SYSTEM temexdmod2
  (* Version 1.0, Author, 4DIAC-Consortium *)
  APPLICATION plantwide
  END_APPLICATION
  APPLICATION App1_ProdQualityandConstraints
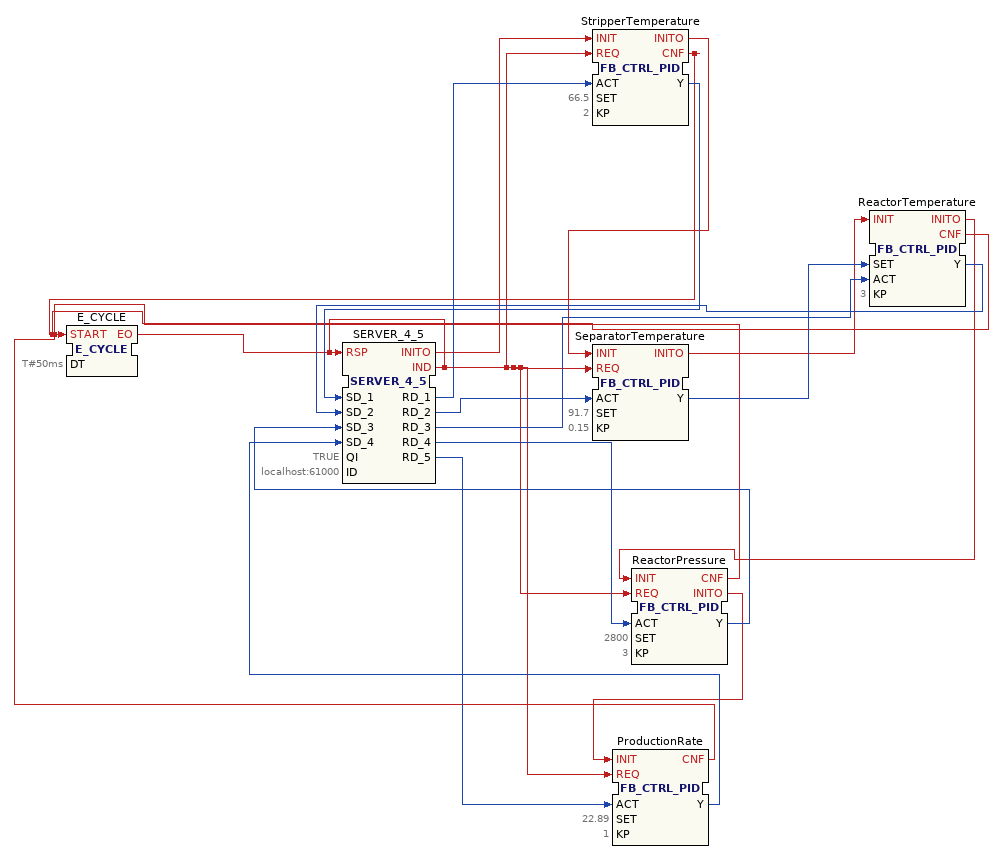
    FBS
      StripperTemperature : FB_CTRL_PID(SET := 66.5, KP := 2);
      ReactorPressure : FB_CTRL_PID(SET := 2800, KP := 3);
      ReactorTemperature : FB_CTRL_PID(KP := 3);
      SeparatorTemperature : FB_CTRL_PID(SET := 91.7, KP := 0.15);
      E_CYCLE : E_CYCLE(DT := T#50ms);
      ProductionRate : FB_CTRL_PID(SET := 22.89, KP := 1);
      SERVER_4_5 : SERVER_4_5(QI := TRUE, ID := localhost:61000);
    END_FBS
    EVENT_CONNECTIONS
      SeparatorTemperature.INITO TO ReactorTemperature.INIT;
      StripperTemperature.INITO TO SeparatorTemperature.INIT;
      ReactorTemperature.INITO TO ReactorPressure.INIT;
      ReactorPressure.CNF TO E_CYCLE.START;
      StripperTemperature.CNF TO E_CYCLE.START;
      ReactorTemperature.CNF TO E_CYCLE.START;
      ReactorPressure.INITO TO ProductionRate.INIT;
      SERVER_4_5.INITO TO StripperTemperature.INIT;
      SERVER_4_5.IND TO StripperTemperature.REQ;
      SERVER_4_5.IND TO SeparatorTemperature.REQ;
      SERVER_4_5.IND TO ReactorPressure.REQ;
      SERVER_4_5.IND TO ProductionRate.REQ;
      ProductionRate.CNF TO E_CYCLE.START;
      E_CYCLE.EO TO SERVER_4_5.RSP;
      SERVER_4_5.IND TO SERVER_4_5.RSP;
    END_CONNECTIONS
    DATA_CONNECTIONS
      SeparatorTemperature.Y TO ReactorTemperature.SET;
      StripperTemperature.Y TO SERVER_4_5.SD_1;
      ReactorTemperature.Y TO SERVER_4_5.SD_2;
      ReactorPressure.Y TO SERVER_4_5.SD_3;
      ProductionRate.Y TO SERVER_4_5.SD_4;
      SERVER_4_5.RD_1 TO StripperTemperature.ACT;
      SERVER_4_5.RD_2 TO SeparatorTemperature.ACT;
      SERVER_4_5.RD_3 TO ReactorTemperature.ACT;
      SERVER_4_5.RD_4 TO ReactorPressure.ACT;
      SERVER_4_5.RD_5 TO ProductionRate.ACT;
    END_CONNECTIONS
  END_APPLICATION
  APPLICATION App2_ControlInventories
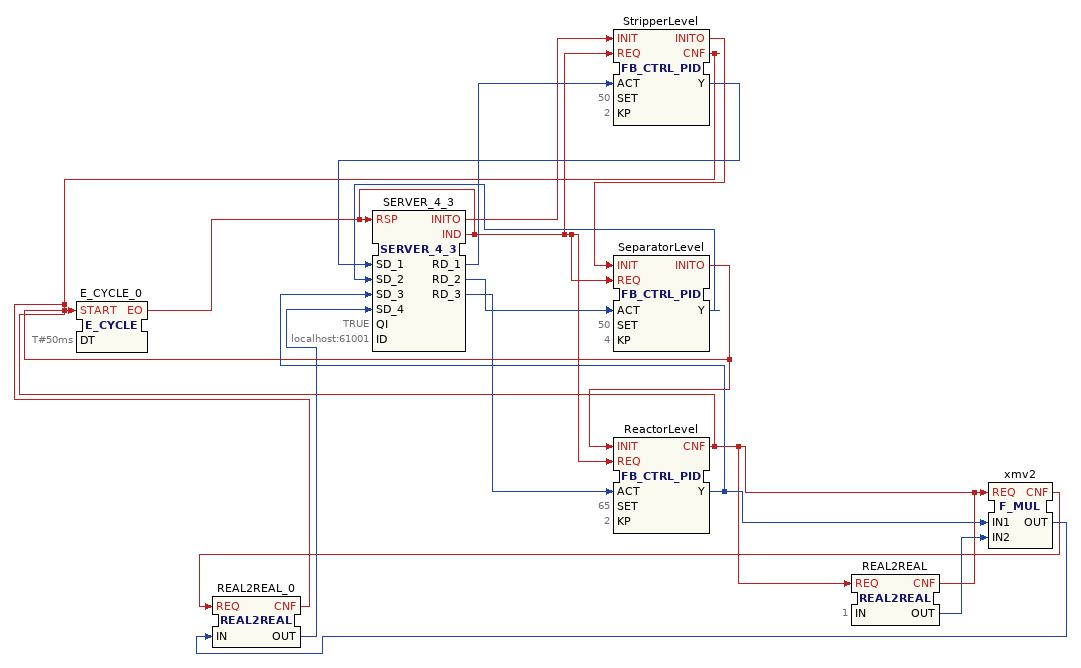
    FBS
      StripperLevel : FB_CTRL_PID(SET := 50, KP := 2);
      SeparatorLevel : FB_CTRL_PID(SET := 50, KP := 4);
      ReactorLevel : FB_CTRL_PID(SET := 65, KP := 2);
      xmv2 : F_MUL;
      REAL2REAL : REAL2REAL(IN := 1);
      E_CYCLE_0 : E_CYCLE(DT := T#50ms);
      SERVER_4_3 : SERVER_4_3(QI := TRUE, ID := localhost:61001);
      REAL2REAL_0 : REAL2REAL;
    END_FBS
    EVENT_CONNECTIONS
      StripperLevel.INITO TO SeparatorLevel.INIT;
      SeparatorLevel.INITO TO ReactorLevel.INIT;
      ReactorLevel.CNF TO REAL2REAL.REQ;
      ReactorLevel.CNF TO xmv2.REQ;
      StripperLevel.CNF TO E_CYCLE_0.START;
      SeparatorLevel.INITO TO E_CYCLE_0.START;
      REAL2REAL.CNF TO xmv2.REQ;
      E_CYCLE_0.EO TO SERVER_4_3.RSP;
      ReactorLevel.CNF TO E_CYCLE_0.START;
      xmv2.CNF TO REAL2REAL_0.REQ;
      REAL2REAL_0.CNF TO E_CYCLE_0.START;
      SERVER_4_3.INITO TO StripperLevel.INIT;
      SERVER_4_3.IND TO StripperLevel.REQ;
      SERVER_4_3.IND TO SeparatorLevel.REQ;
      SERVER_4_3.IND TO ReactorLevel.REQ;
      SERVER_4_3.IND TO SERVER_4_3.RSP;
    END_CONNECTIONS
    DATA_CONNECTIONS
      ReactorLevel.Y TO xmv2.IN1;
      REAL2REAL.OUT TO xmv2.IN2;
      SERVER_4_3.RD_1 TO StripperLevel.ACT;
      SERVER_4_3.RD_2 TO SeparatorLevel.ACT;
      SERVER_4_3.RD_3 TO ReactorLevel.ACT;
      StripperLevel.Y TO SERVER_4_3.SD_1;
      SeparatorLevel.Y TO SERVER_4_3.SD_2;
      ReactorLevel.Y TO SERVER_4_3.SD_3;
      xmv2.OUT TO REAL2REAL_0.IN;
      REAL2REAL_0.OUT TO SERVER_4_3.SD_4;
    END_CONNECTIONS
  END_APPLICATION
  APPLICATION App3_ComponentBalances
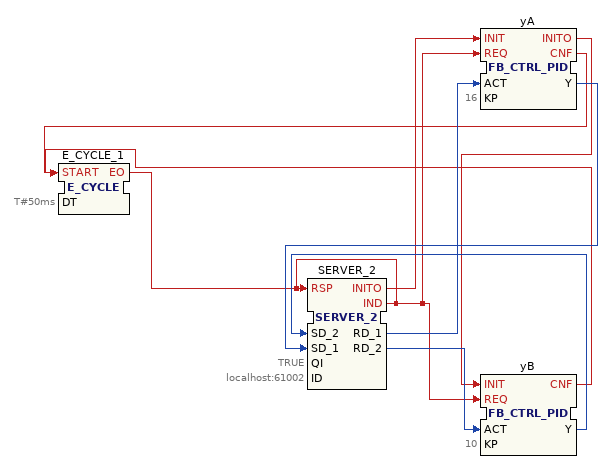
    FBS
      yA : FB_CTRL_PID(KP := 16);
      yB : FB_CTRL_PID(KP := 10);
      SERVER_2 : SERVER_2(QI := TRUE, ID := localhost:61002);
      E_CYCLE_1 : E_CYCLE(DT := T#50ms);
    END_FBS
    EVENT_CONNECTIONS
      yA.INITO TO yB.INIT;
      E_CYCLE_1.EO TO SERVER_2.RSP;
      SERVER_2.INITO TO yA.INIT;
      SERVER_2.IND TO yA.REQ;
      SERVER_2.IND TO yB.REQ;
      yA.CNF TO E_CYCLE_1.START;
      yB.CNF TO E_CYCLE_1.START;
      SERVER_2.IND TO SERVER_2.RSP;
    END_CONNECTIONS
    DATA_CONNECTIONS
      SERVER_2.RD_1 TO yA.ACT;
      SERVER_2.RD_2 TO yB.ACT;
      yB.Y TO SERVER_2.SD_2;
      yA.Y TO SERVER_2.SD_1;
    END_CONNECTIONS
  END_APPLICATION
  DEVICE FORTE_PC : FORTE_PC(MGR_ID := "localhost:61499")
    {SET_ATTRIBUTE(Profile, HOLOBLOC)}
    RESOURCE EMB_RES : EMB_RES
    END_RESOURCE
  END_DEVICE
  SEGMENTS
    Ethernet : Ethernet;
  END_SEGMENTS
  LINKS
    FORTE_PC => Ethernet;
  END_LINKS
END_SYSTEM
